// TIA Portal V20 export
DATA_BLOCK "Runtime_DB"   // DB7
// stored: InstanceOfName Runtime, InstanceOfType FB
"Runtime"
   // VAR_INPUT
   //    "iMotor Run Freedback" : Bool;
   //    iTakt_1Sec : Bool;
   //    iReset : Bool;
   //    iSetTime : Bool;
   // END_VAR
   // VAR_IN_OUT
   //    ioRun_Time_C : "UDT_RunTime_Steuern";
   //    ioRun_Time_S : "UDT_RunTime_Status";
   //    "ioReset_timer-Entern" : Bool;
   // END_VAR
   // VAR
   //    sMotoris_Enabled : Bool;
   //    P_TRIG : Bool;
   // END_VAR
BEGIN
END_DATA_BLOCK
